(* PLC project tni_clock_2, Dassault Systèmes ControlBuild 2024x Refresh1 *)
(* stored: creationDateTime 2024-03-18T18:01:40-01:00 *)

FUNCTION_BLOCK displaymanagement
  VAR_INPUT
    hh : BOOL := false;
    mn : BOOL := false;
    sec : BOOL := false;
    tick : BOOL := false;
    pressure : INT := 0;
  END_VAR
  VAR_IN_OUT
    B1 : BOOL := false;
    B2 : BOOL := false;
    B3 : BOOL := false;
    B4 : BOOL := false;
    displayTime : REAL := 0.0;
    lampSwitchOnTime : REAL := 0.0;
    pulseTime : INT := 0;
  END_VAR
  VAR_OUTPUT
    displayValue : BOOL := false;
    switchOnLight : BOOL := false;
  END_VAR


ACTION C_source_code:

END_ACTION
END_FUNCTION_BLOCK

FUNCTION_BLOCK timemanagement
  VAR_INPUT
    tick : BOOL := false;
  END_VAR
  VAR_IN_OUT
    B1 : BOOL := false;
    B2 : BOOL := false;
    B3 : BOOL := false;
    B4 : BOOL := false;
    tickCount : REAL := 0.0;
    adjustMode : INT := 0;
  END_VAR
  VAR_OUTPUT
    stepMotorSecond : BOOL := false;
    stepMotorMinute : BOOL := false;
    stepMotorHour : BOOL := false;
    hh : BOOL := false;
    mn : BOOL := false;
    sec : BOOL := false;
  END_VAR


ACTION C_source_code:

END_ACTION
END_FUNCTION_BLOCK

PROGRAM controller
  VAR_INPUT
    pressure : INT := 0;
    tick : BOOL := false;
  END_VAR
  VAR_IN_OUT
    B1 : BOOL := false;
    B2 : BOOL := false;
    B3 : BOOL := false;
    B4 : BOOL := false;
  END_VAR
  VAR_OUTPUT
    displayValue : BOOL := false;
    stepMotorSecond : BOOL := false;
    stepMotorMinute : BOOL := false;
    stepMotorHour : BOOL := false;
    switchOnLight : BOOL := false;
  END_VAR

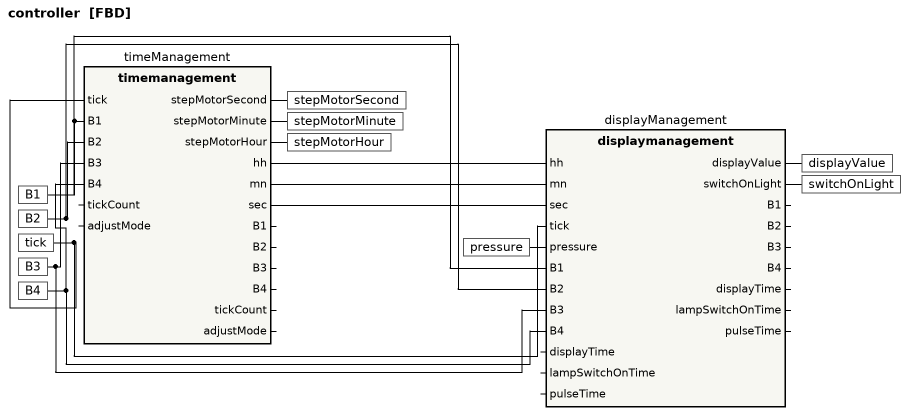
(* FBD diagram, written out as Structured Text *)
timeManagement(tick := tick, B1 := B1, B2 := B2, B3 := B3, B4 := B4);
displayManagement(hh := timeManagement.hh, mn := timeManagement.mn, sec := timeManagement.sec, tick := tick, pressure := pressure, B1 := B1, B2 := B2, B3 := B3, B4 := B4);
displayValue := displayManagement.displayValue;
stepMotorSecond := timeManagement.stepMotorSecond;
stepMotorMinute := timeManagement.stepMotorMinute;
stepMotorHour := timeManagement.stepMotorHour;
switchOnLight := displayManagement.switchOnLight;
END_PROGRAM

FUNCTION_BLOCK environment
  VAR_INPUT
    depth : INT := 0;
  END_VAR
  VAR_IN_OUT
    B1 : BOOL := false;
    B2 : BOOL := false;
    B3 : BOOL := false;
    B4 : BOOL := false;
    hydrostaticPressure : REAL := 0.0;
    absolutePressure : REAL := 0.0;
  END_VAR
  VAR_OUTPUT
    pressure : INT := 0;
    tick : BOOL := false;
  END_VAR


ACTION C_source_code:

END_ACTION
END_FUNCTION_BLOCK

FUNCTION_BLOCK lcd
  VAR_INPUT
    displayValue : BOOL := false;
  END_VAR
  VAR_IN_OUT
    displayString : BOOL := false;
    i : BOOL := false;
  END_VAR


ACTION C_source_code:

END_ACTION
END_FUNCTION_BLOCK

FUNCTION_BLOCK light
  VAR_INPUT
    switchOnLight : BOOL := false;
  END_VAR


ACTION C_source_code:

END_ACTION
END_FUNCTION_BLOCK

FUNCTION_BLOCK motors
  VAR_INPUT
    stepMotorSecond : BOOL := false;
    stepMotorMinute : BOOL := false;
    stepMotorHour : BOOL := false;
  END_VAR
  VAR_IN_OUT
    hourHand : INT := 0;
    minuteHand : INT := 0;
    secondHand : INT := 0;
  END_VAR


ACTION C_source_code:

END_ACTION
END_FUNCTION_BLOCK

PROGRAM my_app.tni_clock_2
  VAR_INPUT
    depth : INT := 0;
  END_VAR
  VAR_IN_OUT
    B1 : BOOL := false;
    B2 : BOOL := false;
    B3 : BOOL := false;
    B4 : BOOL := false;
  END_VAR

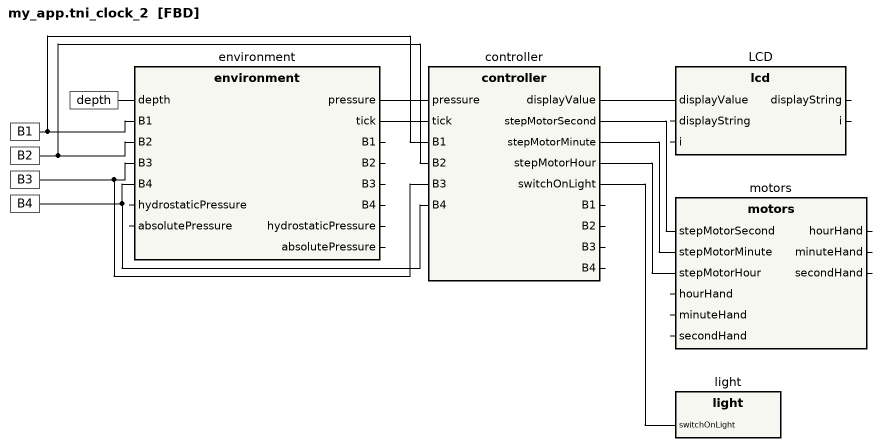
(* FBD diagram, written out as Structured Text *)
environment(depth := depth, B1 := B1, B2 := B2, B3 := B3, B4 := B4);
controller(pressure := environment.pressure, tick := environment.tick, B1 := B1, B2 := B2, B3 := B3, B4 := B4);
LCD(displayValue := controller.displayValue);
motors(stepMotorSecond := controller.stepMotorSecond, stepMotorMinute := controller.stepMotorMinute, stepMotorHour := controller.stepMotorHour);
light(switchOnLight := controller.switchOnLight);
END_PROGRAM
